FUNCTION Convert_DATE_TO_USINT : Hresult
VAR_INPUT
	in : DATE;
	out : REFERENCE TO USINT;
END_VAR
VAR
	converted : USINT;
END_VAR
VAR CONSTANT
	INCOMPATIBLE : HRESULT := 16#9811070E;
END_VAR

converted := DATE_TO_USINT(in);

IF (USINT_TO_DATE(converted) <> in) THEN
	Convert_DATE_TO_USINT := INCOMPATIBLE;
	RETURN;
END_IF

out := converted;

END_FUNCTION

(* stored: Version 1.1.0.1, ProductVersion 3.1.4024.12
   POU Convert_DATE_TO_USINT: Id {d256960a-e1f9-4199-afdc-6647f12d62bf}, SpecialFunc None *)
